FUNCTION_BLOCK OF_E_R_TRIG (* Boolean rising edge detection *)
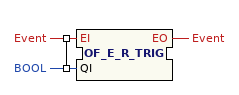
  EVENT_INPUT
    EI WITH QI; (* check for rising edge *)
  END_EVENT
  EVENT_OUTPUT
    EO; (* confirmation that an rising edge was detected *)
  END_EVENT
  VAR_INPUT
    QI : BOOL; (* value to check for a rising edge *)
  END_VAR
END_FUNCTION_BLOCK
